(* PLC project Exercise1, ExampleCompany OpenPLC 1.0 *)
(* stored: creationDateTime 2024-05-15T20:23:44.2566394, modificationDateTime 2024-05-15T20:23:18.1300557 *)

PROGRAM MainProgram
  VAR
    A : REAL;
    B : REAL;
    C : REAL;
    Avg : REAL;
  END_VAR

            Avg := (A + B + C) / 3;
          
END_PROGRAM
